{attribute 'qualified_only'}
VAR_GLOBAL
	Inputs	:	ARRAY[0..255] OF WORD;		//入力レジスタModbusマスター読み取りのみ
	Outputs :	ARRAY[0..255] OF WORD;		//保持レジスタModbusマスター読み書き可能
	Memory 	:	ARRAY[0..255] OF WORD;		//Modbusマスター読み書き可能
END_VAR

(* stored: Version 1.1.0.1
   GVL GVL_SerialCom: Id {94fe65de-c7e4-479f-a19f-56f48dfce30d} *)
